FUNCTION_BLOCK FB_Closedloop
VAR_INPUT
END_VAR
VAR_OUTPUT
END_VAR
VAR
END_VAR

END_FUNCTION_BLOCK

(* stored: Version 1.1.0.1, ProductVersion 3.1.4024.12
   POU FB_Closedloop: Id {0a291c2b-edcc-4387-9508-1fc34f82f1c8}, SpecialFunc None *)
